// TIA Portal project "AWL LIBRO 2" (V11)

(* hardware
DEVICE "S7300/ET200 station_1"  SIMATIC 300-Station
   slot 0: "Perfil soporte_0"  Rail  6ES7 390-1***0-0AA0
   slot 2: "PLC_1"  CPU 313C-2 DP  6ES7 313-6CF03-0AB0  V2.6
      slot 0: "Interfaz MPI_1"  MPI
      slot 1: "Interfaz DP_1"  DP
      slot 2: "DI16/DO16_1"  DI16/DO16
      slot 4: "Contaje_1"  Counter
*)

// ===== PLC "PLC_1"  CPU 313C-2 DP =====

VAR_GLOBAL   // PLC tag table "Tabla de variables estándar"
   "PARO" AT %E0.0 : Bool;
   "MARCHA" AT %E0.1 : Bool;
   "MOTOR 1" AT %A0.0 : Bool;
   "LED 1" AT %A0.1 : Bool;
   "MOTOR 2" AT %A0.2 : Bool;
   "LED 2" AT %A0.3 : Bool;
   "LED PARO" AT %A0.4 : Bool;
   "LED AVERIA" AT %A0.5 : Bool;
   "Tag_1" AT %M10.0 : Bool;
   "Tag_2" AT %M10.1 : Bool;
   "SALIDAS" AT %AB0 : Byte;
   "Tag_4" AT %M10.2 : Bool;
   "Tag_5" AT %T0 : Timer;
   "Tag_3" AT %T1 : Timer;
   "Tag_6" AT %M10.3 : Bool;
   "Tag_7" AT %E0.3 : Bool;
   "RELE TERMICO" AT %E0.2 : Bool;
   "Tag_8" AT %M10.4 : Bool;
END_VAR

ORGANIZATION_BLOCK "Main"   // OB1, STL
TITLE = EJERCICO 2 LIBRO / "Main Program Sweep (Cycle)"
{ S7_Optimized_Access := 'FALSE' }
VERSION : 0.1
   VAR_TEMP
      OB1_EV_CLASS : Byte;   // Bits 0-3 = 1 (Coming event), Bits 4-7 = 1 (Event class 1)
      OB1_SCAN_1 : Byte;   // 1 (Cold restart scan 1 of OB 1), 3 (Scan 2-n of OB 1)
      OB1_PRIORITY : Byte;   // Priority of OB Execution
      OB1_OB_NUMBR : Byte;   // 1 (Organization block 1, OB1)
      OB1_RESERVED_1 : Byte;   // Reserved for system
      OB1_RESERVED_2 : Byte;   // Reserved for system
      OB1_PREV_CYCLE : Int;   // Cycle time of previous OB1 scan (milliseconds)
      OB1_MIN_CYCLE : Int;   // Minimum cycle time of OB1 (milliseconds)
      OB1_MAX_CYCLE : Int;   // Maximum cycle time of OB1 (milliseconds)
      OB1_DATE_TIME : Date_And_Time;   // Date and time OB1 started
   END_VAR
BEGIN

REGION Network 1
         AN    "Tag_1";  // REPOSO LED PARO ENCENDIDO.
         FP    "Tag_2";
         JNB   _001;
         L     B#16#10;
         T     "SALIDAS";
   _001: NOP   0;
         O     "MARCHA";  // ARRANQUE MOTOR 1 Y LED 1.
         O     "Tag_3";  // CONTACTO T1 CICLICO.
         FP    "Tag_4";
         JNB   _002;
         L     B#16#3;
         T     "SALIDAS";
   _002: NOP   0;
         A     "MOTOR 1";  // TEMOPORIZADO 3S CAMBIO DE MOTOR.
         L     S5T#3S;
         SD    "Tag_5";
         A     "Tag_5";
         JNB   _003;
         L     B#16#C;
         T     "SALIDAS";
   _003: NOP   0;
         A     "MOTOR 2";  // TEMPORIZADO 2S CAMBIO DE MOTOR.
         L     S5T#2S;
         SD    "Tag_3";
         A     "PARO";  // PARO DE SECUENCIA POSICION DE REPOSO.
         FP    "Tag_6";
         JNB   _004;
         L     B#16#10;
         T     "SALIDAS";
   _004: NOP   0;
         A     "RELE TERMICO";  // DISPARO TERMICO.
         JNB   _005;
         L     B#16#30;
         T     "SALIDAS";
   _005: NOP   0;
         A     "RELE TERMICO";
         FN    "Tag_8";
         JNB   _006;
         L     B#16#10;
         T     "SALIDAS";
   _006: NOP   0;
END_REGION
END_ORGANIZATION_BLOCK